{attribute 'qualified_only'}
{attribute 'strict'}
TYPE GripperCmd :
(
	noGrip ,
	take ,
	put  
);
END_TYPE

(* stored: Version 1.1.0.1, ProductVersion 3.1.4024.11
   DUT GripperCmd: Id {a6af5599-df13-4a0d-ab06-61e21ff7d27a} *)
